FUNCTION_BLOCK fbSliderWithGripperEM EXTENDS fbEM

// TEST
em.Config.Data.Q[10] := true;

END_FUNCTION_BLOCK

(* stored: Version 1.1.0.1, ProductVersion 3.1.4024.12
   POU fbSliderWithGripperEM: Id {262a0099-d26a-4a20-85d1-5e68be47c9f0}, SpecialFunc None *)
